// TIA Portal V19 export
TYPE "LAF_typeConstraintRollerEm2Parameters"
// stored: Access Published
   STRUCT
      cm1Vfd206 : "LAF_typeVfdParameters";
      cm5Axis107 { S7_SetPoint := 'True'} : "LAF_typeAxisParameters";
      cm8Scanner { S7_SetPoint := 'True'} : "LAF_typeSR1000Parameters";
   END_STRUCT;
END_TYPE
